FUNCTION_BLOCK FB_Servo

(*
	Beckhoff motion
*)

VAR_INPUT
	stAxis:			AXIS_REF;
	
	fOverride:		LREAL;
	
END_VAR

VAR_OUTPUT
END_VAR

VAR
// instance data
	fbPower:		MC_POWER;

END_VAR




// MC_POWER
fbPower(
	Axis:= stAxis, 
	Enable:= TRUE, 
	Enable_Positive:= TRUE, 
	Enable_Negative:= TRUE, 
	Override:= fOverride, 
	BufferMode:= , 
	Options:= , 
	Status=> , 
	Busy=> , 
	Active=> , 
	Error=> , 
	ErrorID=> );

END_FUNCTION_BLOCK

(* stored: Version 1.1.0.1, ProductVersion 3.1.4024.4
   POU FB_Servo: Id {8f67c982-b1b7-4ac1-80c7-dec324316813}, SpecialFunc None *)
